PROGRAM MAIN
VAR
	fbJson:FB_JsonSaxWriter;
	fbJsonDomParser:FB_JsonDomParser;

	fbSaveFile :FB_SaveFile;
	fbReadJsonReal :FB_ReadJsonReal;
	
	jsonDOC : SJsonValue;
	
	Trigger: BOOL:=TRUE;
	sBuffer :STRING(100);
	r32:REAL;

	bSave:BOOL;

	
	bLoadJsonFile:BOOL;
	jSonProp :SJsonValue;
	jsonRoot :SJsonValue;
	fSensorValue :LREAL;
	bReadValue:BOOL;
END_VAR


IF Trigger THEN
	r32:=r32+0.01;
	IF r32>=1000.0 THEN
		r32:=0.0;
	END_IF

	//Object creation
	fbJson.StartObject(); //Open Bracket
		fbJson.AddKey('Sensor1');
		fbJson.AddReal((r32));
	fbJson.EndObject(); //Close Bracket
	
	//Document creation
	sBuffer := fbJson.GetDocument();
	fbJson.ResetDocument();
	
END_IF

//Save information
IF bSave THEN
	fbSaveFile(sPath:='C:\TwinCAT\3.1\Boot\MyData.json',AmsNetId:='',sBuffer:=sBuffer);
	bSave:=FALSE;
END_IF

//Read information
IF bLoadJsonFile THEN
fbReadJsonReal(Member:='Sensor1',sPath:='C:\TwinCAT\3.1\Boot\MyData.json',fReadValue=>);
fSensorValue:= fbReadJsonReal.fReadValue;
END_IF

END_PROGRAM

(* stored: Version 1.1.0.1, ProductVersion 3.1.4024.14
   POU MAIN: Id {81fdac0f-1e0d-486a-ba31-7d84129b3f10}, SpecialFunc None *)
